//{attribute 'qualified_only'}
VAR_GLOBAL
	bMotorScreen1Omhoog		AT %Q*: BOOL;
	bMotorScreen1Omlaag		AT %Q*: BOOL;
	bMotorScreen2Omhoog		AT %Q*: BOOL;
	bMotorScreen2Omlaag		AT %Q*: BOOL;
	bMotorScreen3Omhoog		AT %Q*: BOOL;
	bMotorScreen3Omlaag		AT %Q*: BOOL;
	bMotorScreen4Omhoog		AT %Q*: BOOL;
	bMotorScreen4Omlaag		AT %Q*: BOOL;

	bMotorRolluik1Omhoog	AT %Q*: BOOL;
	bMotorRolluik1Omlaag	AT %Q*: BOOL;
	bMotorRolluik2Omhoog	AT %Q*: BOOL;
	bMotorRolluik2Omlaag	AT %Q*: BOOL;
	bMotorRolluik3Omhoog	AT %Q*: BOOL;
	bMotorRolluik3Omlaag	AT %Q*: BOOL;
END_VAR

(* stored: Version 1.1.0.1
   GVL GVL_Screens: Id {06ff7f98-a7d1-4ca6-98ac-40bfa1f24541} *)
